Omron CX-Programmer project NewProject (CX-Programmer 9.61)

# PLC NewPLC1: CP1E N30

## Global symbols (name address type ; comment)
0.00 BOOL  ; PB1
0.01 BOOL  ; RESET
100.00 BOOL  ; LED
T000 BOOL  ; TIMER1

## Program NewProgram1 (cyclic task 0)

### Section Section1

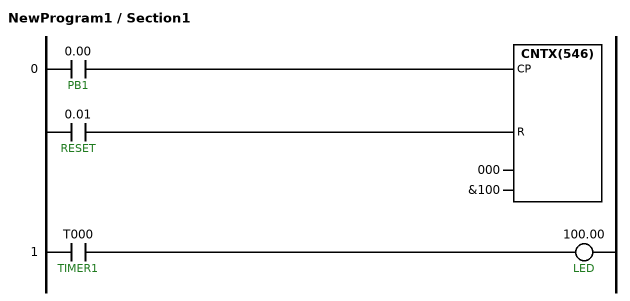
; rung 0
LD 0.00  ; PB1
LD 0.01  ; RESET
CNTX(546) 000 &100
; rung 1
LD T000  ; TIMER1
OUT 100.00  ; LED

### Section END
; rung 0
END(001)